# EPICS substitutions: iocs/newportIOC/iocBoot/iocNewport/ESP300.substitutions
file "$(MOTOR)/db/motor.db"
{
pattern
{P,         N,        M,      DTYP,    C,  S,  DESC,          EGU,      DIR,  VELO,  VBAS,  ACCL,  BDST,  BVEL,  BACC,  MRES,  PREC,  DHLM,  DLLM,  INIT}
{newport:,  21,   "m$(N)",  "ESP300",  0,  0,  "motor $(N)",  mm,       Pos,  1,     .1,    .2,    0,     1,     .2,    5e-5,  5,     100,   -100,  ""}
{newport:,  22,   "m$(N)",  "ESP300",  0,  1,  "motor $(N)",  mm,       Pos,  1,     .1,    .2,    0,     1,     .2,    5e-5,  5,     100,   -100,  ""}
{newport:,  23,   "m$(N)",  "ESP300",  0,  2,  "motor $(N)",  mm,       Pos,  1,     .1,    .2,    0,     1,     .2,    5e-5,  5,     100,   -100,  ""}
}
